(* IEC 61131-3 sources: AXOpen/src/components.rexroth.drives/ctrl/src/AxoCtrlxDriveXsc (part 4) *)

                IF _State>=UINT#430 AND _State<UINT#437 THEN
                    IF _AxisReference^.Data.Cycle <> MC_ReadBoolParameterCycle THEN
                        _AxisReference^.Data.Cycle := _AxisReference^.Data.Cycle - ULINT#1;
                        _State := UINT#439;
                    END_IF;
                END_IF;
            END_IF;

            IF NOT Enable AND MC_ReadBoolParameterEnable_PV AND _State>=UINT#430 AND _State<=UINT#439 THEN
                _AxisReference^.Status.CurrentMotionTaskId := AXOpen.Components.Drives.eAxoMotionTaskId#Axo_None;
                MC_ReadBoolParameterErrorID := WORD#0;
                MC_ReadBoolParameterCycle := ULINT#0;
                MC_ReadBoolParameterValid := FALSE;
                MC_ReadBoolParameterValue := FALSE;
                _State := UINT#0;
            END_IF;

            ErrorID := TO_DINT(MC_ReadBoolParameterErrorID);
            Valid := MC_ReadBoolParameterValid;
            Value := MC_ReadBoolParameterValue;
            MC_ReadBoolParameterEnable_PV := Enable;

        END_METHOD

        ///<summary>
        /// This method modifies the value of a vendor specific parameter.
        ///</summary>
        VAR INTERNAL
            MC_WriteParameterExecute_PV     : 	BOOL := FALSE;		//Enable - previous value
            MC_WriteParameterErrorID        : 	WORD;
            MC_WriteParameterCycle			: 	ULINT;
        END_VAR
        METHOD PUBLIC OVERRIDE MC_WriteParameter
            VAR_INPUT
                AxisRef         :   AXOpen.Components.Abstractions.Drives.IAxoAxisReference;
                Execute         :   BOOL;                       //  Write the value of the parameter at rising edge
                ParameterNumber :   DINT;                       //  Number of the parameter (correspondence between number andparameter is specified in the table above)
                Value           :   LINT;                       //  New value of the specified parameter
                ExecutionMode   :   AXOpen.Components.Abstractions.Drives.eAxoExecutionMode;          //  Defines the chronological sequence of the method.
            END_VAR
            VAR_OUTPUT
                Done            :   BOOL;                       //  Parameter successfully written
                Busy            :   BOOL;                       //  The method is not finished and new output values are to be expected.
                Error           :   BOOL;                       //  Signals that an error has occurred within the method
                ErrorID         :   DINT;                       //  Error identification
            END_VAR
            VAR
                _AxisReference :  REF_TO AXOpen.Components.Rexroth.Drives.AxoCtrlxDriveXscAxisReference;
            END_VAR

            _AxisReference ?= AxisRef;

            IF(_AxisReference = NULL) THEN
                Messenger.Activate(     UINT#1610, eAxoMessageCategory#ProgrammingError);
                DriveStatus.Error.Id := UINT#1610;
                RETURN;
            END_IF;

            IF THIS.AxoWriteParameter_Task.StartTriggered()  THEN
                _AxisReference^.Status.CurrentMotionTaskId := AXOpen.Components.Drives.eAxoMotionTaskId#Axo_WriteParameter;
            END_IF;

            IF Execute AND NOT MC_WriteParameterExecute_PV AND _State = UINT#0 THEN
                _AxisReference^.Data.Cycle := _AxisReference^.Data.Cycle + ULINT#2;
                MC_WriteParameterCycle := _AxisReference^.Data.Cycle ;
            END_IF;

            IF Execute THEN
                IF _State = UINT#0 THEN
                    Busy := TRUE;
                    THIS.CallTimers(FALSE);
                    DriveStatus.Error.Id :=  UINT#0;
                    TaskMessenger.Restore();
                    _State := UINT#440;
                END_IF;
                IF _State = UINT#440 THEN
                    IF _infoTimer.output THEN
                        TaskMessenger.Activate( UINT#640, eAxoMessageCategory#Potential);
                        DriveStatus.Error.Id := UINT#640;
                    END_IF;
                    Busy := TRUE;
                    _lword :=  TO_LWORD(Value);
                    _data8[0] := _lword.%B0;
                    _data8[1] := _lword.%B1;
                    _data8[2] := _lword.%B2;
                    _data8[3] := _lword.%B3;
                    _data8[4] := _lword.%B4;
                    _data8[5] := _lword.%B5;
                    _data8[6] := _lword.%B6;
                    _data8[7] := _lword.%B7;
                    _WriteRecord(   request     :=  TRUE,
                                    hardwareID  :=  (AxisRefExt.HWIDs.HW_S_0_0134_0_0),
                                    index       :=  ParameterNumber,
                                    length      :=  UINT#8,
                                    record      :=  _data8);
                    IF NOT _WriteRecord.busy AND _WriteRecord.done AND NOT _WriteRecord.error THEN
                        _State := UINT#441;
                    ElSIF _WriteRecord.error THEN
                        _WriteRecord(request := FALSE, record := _data8);
                        Messenger.Activate(         UINT#1611, eAxoMessageCategory#Error);
                        MC_WriteParameterErrorID := WORD#1611;
                        _State := UINT#449;
                    END_IF;
                END_IF;
                IF _State = UINT#441 THEN
                    _WriteRecord(request := FALSE, record := _data8);
                    IF NOT _WriteRecord.busy AND NOT _WriteRecord.done AND NOT _WriteRecord.error  THEN
                        _State := UINT#447;
                    END_IF;
                END_IF;
                IF _State = UINT#447 THEN
                    Done := TRUE;
                    MC_WriteParameterCycle := ULINT#0;
                END_IF;
                IF _State = UINT#449 THEN
                    MC_WriteParameterCycle := ULINT#0;
                    Error := TRUE;
                END_IF;

                IF _State>=UINT#440 AND _State<UINT#447 THEN
                    IF _AxisReference^.Data.Cycle <> MC_WriteParameterCycle THEN
                        _AxisReference^.Data.Cycle := _AxisReference^.Data.Cycle - ULINT#1;
                        _State := UINT#449;
                    END_IF;
                END_IF;
            END_IF;

            IF THIS.AxoWriteParameter_Task.DoneReached() AND _State>=UINT#440 AND _State<=UINT#449 THEN
                _AxisReference^.Status.CurrentMotionTaskId := AXOpen.Components.Drives.eAxoMotionTaskId#Axo_Done;
                MC_WriteParameterErrorID := WORD#0;
                // MC_WriteParameterCycle := ULINT#0;
                _State := UINT#0;
            END_IF;

            IF THIS.AxoWriteParameter_Task.RestoreTriggered() AND _State>=UINT#440 AND _State<=UINT#449 THEN
                _AxisReference^.Status.CurrentMotionTaskId := AXOpen.Components.Drives.eAxoMotionTaskId#Axo_None;
                MC_WriteParameterErrorID := WORD#0;
                MC_WriteParameterCycle := ULINT#0;
                _State := UINT#0;
            END_IF;

            ErrorID := TO_DINT(MC_WriteParameterErrorID);
            MC_WriteParameterExecute_PV := Execute;
        END_METHOD

        ///<summary>
        /// This method modifies the value of a vendor specific parameter of type Real.
        ///</summary>
        VAR INTERNAL
            MC_WriteRealParameterExecute_PV     : 	BOOL := FALSE;		//Enable - previous value
            MC_WriteRealParameterErrorID        : 	WORD;
            MC_WriteRealParameterCycle			: 	ULINT;
        END_VAR
        METHOD PUBLIC OVERRIDE MC_WriteRealParameter
            VAR_INPUT
                AxisRef         :   AXOpen.Components.Abstractions.Drives.IAxoAxisReference;
                Execute         :   BOOL;                       //  Write the value of the parameter at rising edge
                ParameterNumber :   DINT;                       //  Number of the parameter (correspondence between number andparameter is specified in the table above)
                Value           :   REAL;                       //  New value of the specified parameter
                ExecutionMode   :   AXOpen.Components.Abstractions.Drives.eAxoExecutionMode;          //  Defines the chronological sequence of the method.
            END_VAR
            VAR_OUTPUT
                Done            :   BOOL;                       //  Parameter successfully written
                Busy            :   BOOL;                       //  The method is not finished and new output values are to be expected.
                Error           :   BOOL;                       //  Signals that an error has occurred within the method
                ErrorID         :   DINT;                       //  Error identification
            END_VAR
            VAR
                _AxisReference :  REF_TO AXOpen.Components.Rexroth.Drives.AxoCtrlxDriveXscAxisReference;
            END_VAR

            _AxisReference ?= AxisRef;

            IF(_AxisReference = NULL) THEN
                Messenger.Activate(     UINT#1620, eAxoMessageCategory#ProgrammingError);
                DriveStatus.Error.Id := UINT#1620;
                RETURN;
            END_IF;

            IF THIS.AxoWriteRealParameter_Task.StartTriggered()  THEN
                _AxisReference^.Status.CurrentMotionTaskId := AXOpen.Components.Drives.eAxoMotionTaskId#Axo_WriteRealParameter;
            END_IF;

            IF Execute AND NOT MC_WriteRealParameterExecute_PV AND _State = UINT#0 THEN
                _AxisReference^.Data.Cycle := _AxisReference^.Data.Cycle + ULINT#2;
                MC_WriteRealParameterCycle := _AxisReference^.Data.Cycle ;
            END_IF;

            IF Execute THEN
                IF _State = UINT#0 THEN
                    Busy := TRUE;
                    _State := UINT#450;
                END_IF;
                IF _State = UINT#450 THEN
                    IF _infoTimer.output THEN
                        TaskMessenger.Activate( UINT#650, eAxoMessageCategory#Potential);
                        DriveStatus.Error.Id := UINT#650;
                    END_IF;
                    Busy := TRUE;
                    _dword :=  TO_DWORD(TO_DINT(Value));
                    _data4[0] := _dword.%B0;
                    _data4[1] := _dword.%B1;
                    _data4[2] := _dword.%B2;
                    _data4[3] := _dword.%B3;
                    _WriteRecord(   request     :=  TRUE,
                                    hardwareID  :=  (AxisRefExt.HWIDs.HW_S_0_0134_0_0),
                                    index       :=  ParameterNumber,
                                    length      :=  UINT#4,
                                    record      :=  _data4);
                    IF NOT _WriteRecord.busy AND _WriteRecord.done AND NOT _WriteRecord.error THEN
                        _State := UINT#451;
                    ElSIF _WriteRecord.error THEN
                        _WriteRecord(request := FALSE, record := _data4);
                        Messenger.Activate(             UINT#1621, eAxoMessageCategory#Error);
                        MC_WriteRealParameterErrorID := WORD#1621;
                        _State := UINT#459;
                    END_IF;
                END_IF;
                IF _State = UINT#451 THEN
                    IF _infoTimer.output THEN
                        TaskMessenger.Activate( UINT#651, eAxoMessageCategory#Potential);
                        DriveStatus.Error.Id := UINT#651;
                    END_IF;
                    Busy := TRUE;
                    _WriteRecord(request := FALSE, record := _data4);
                    IF NOT _WriteRecord.busy AND NOT _WriteRecord.done AND NOT _WriteRecord.error THEN
                        _State := UINT#457;
                    END_IF;
                END_IF;
                IF _State = UINT#457 THEN
                    Done := TRUE;
                    MC_WriteRealParameterCycle := ULINT#0;
                END_IF;
                IF _State = UINT#459 THEN
                    MC_WriteRealParameterCycle := ULINT#0;
                    Error := TRUE;
                END_IF;

                IF _State>=UINT#450 AND _State<UINT#457 THEN
                    IF _AxisReference^.Data.Cycle <> MC_WriteRealParameterCycle THEN
                        _AxisReference^.Data.Cycle := _AxisReference^.Data.Cycle - ULINT#1;
                        _State := UINT#459;
                    END_IF;
                END_IF;
            END_IF;

            IF THIS.AxoWriteRealParameter_Task.DoneReached() AND _State>=UINT#450 AND _State<=UINT#459 THEN
                _AxisReference^.Status.CurrentMotionTaskId := AXOpen.Components.Drives.eAxoMotionTaskId#Axo_Done;
                MC_WriteRealParameterErrorID := WORD#0;
                // MC_WriteRealParameterCycle := ULINT#0;
                _State := UINT#0;
            END_IF;

            IF THIS.AxoWriteRealParameter_Task.RestoreTriggered() AND _State>=UINT#450 AND _State<=UINT#459 THEN
                _AxisReference^.Status.CurrentMotionTaskId := AXOpen.Components.Drives.eAxoMotionTaskId#Axo_None;
                MC_WriteRealParameterErrorID := WORD#0;
                MC_WriteRealParameterCycle := ULINT#0;
                _State := UINT#0;
            END_IF;

            ErrorID := TO_DINT(MC_WriteRealParameterErrorID);
            MC_WriteRealParameterExecute_PV := Execute;
        END_METHOD

        ///<summary>
        /// This method modifies the value of a vendor specific parameter of type BOOL.
        ///</summary>
        VAR INTERNAL
            MC_WriteBoolParameterExecute_PV     : 	BOOL := FALSE;		//Enable - previous value
            MC_WriteBoolParameterErrorID        : 	WORD;
            MC_WriteBoolParameterCycle			: 	ULINT;
        END_VAR
        METHOD PUBLIC OVERRIDE MC_WriteBoolParameter
            VAR_INPUT
                AxisRef         :   AXOpen.Components.Abstractions.Drives.IAxoAxisReference;
                Execute         :   BOOL;                       //  Write the value of the parameter at rising edge
                ParameterNumber :   DINT;                       //  Number of the parameter (correspondence between number andparameter is specified in the table above)
                Value           :   BOOL;                       //  New value of the specified parameter
                ExecutionMode   :   AXOpen.Components.Abstractions.Drives.eAxoExecutionMode;          //  Defines the chronological sequence of the method.
            END_VAR
            VAR_OUTPUT
                Done            :   BOOL;                       //  Parameter successfully written
                Busy            :   BOOL;                       //  The method is not finished and new output values are to be expected.
                Error           :   BOOL;                       //  Signals that an error has occurred within the method
                ErrorID         :   DINT;                       //  Error identification
            END_VAR
            VAR
                _AxisReference :  REF_TO AXOpen.Components.Rexroth.Drives.AxoCtrlxDriveXscAxisReference;
            END_VAR

            _AxisReference ?= AxisRef;

            IF(_AxisReference = NULL) THEN
                Messenger.Activate(     UINT#1630, eAxoMessageCategory#ProgrammingError);
                DriveStatus.Error.Id := UINT#1630;
                RETURN;
            END_IF;

            IF THIS.AxoWriteBoolParameter_Task.StartTriggered()  THEN
                _AxisReference^.Status.CurrentMotionTaskId := AXOpen.Components.Drives.eAxoMotionTaskId#Axo_WriteBoolParameter;
            END_IF;

            IF Execute AND NOT MC_WriteBoolParameterExecute_PV AND _State = UINT#0 THEN
                _AxisReference^.Data.Cycle := _AxisReference^.Data.Cycle + ULINT#2;
                MC_WriteBoolParameterCycle := _AxisReference^.Data.Cycle ;
            END_IF;

            IF Execute THEN
                IF _State = UINT#0 THEN
                    Busy := TRUE;
                    _State := UINT#460;
                END_IF;
                IF _State = UINT#460 THEN
                    IF _infoTimer.output THEN
                        TaskMessenger.Activate( UINT#660, eAxoMessageCategory#Potential);
                        DriveStatus.Error.Id := UINT#660;
                    END_IF;
                    Busy := TRUE;
                    _dword :=  TO_DWORD(TO_DINT(Value));
                    _data2[0].%X0 := Value;
                    _WriteRecord(   request     :=  TRUE,
                                    hardwareID  :=  (AxisRefExt.HWIDs.HW_S_0_0134_0_0),
                                    index       :=  ParameterNumber,
                                    length      :=  UINT#2,
                                    record      :=  _data2);
                    IF NOT _WriteRecord.busy AND _WriteRecord.done AND NOT _WriteRecord.error THEN
                        _State := UINT#461;
                    ElSIF _WriteRecord.error THEN
                        _WriteRecord(request := FALSE, record := _data2);
                        Messenger.Activate(             UINT#1631, eAxoMessageCategory#Error);
                        MC_WriteBoolParameterErrorID := WORD#1631;
                        _State := UINT#469;
                    END_IF;
                END_IF;
                IF _State = UINT#461 THEN
                    IF _infoTimer.output THEN
                        TaskMessenger.Activate( UINT#661, eAxoMessageCategory#Potential);
                        DriveStatus.Error.Id := UINT#661;
                    END_IF;
                    Busy := TRUE;
                    _WriteRecord(request := FALSE, record := _data2);
                    IF NOT _WriteRecord.busy AND _WriteRecord.done AND NOT _WriteRecord.error THEN
                        _State := UINT#467;
                    END_IF;
                END_IF;
                IF _State = UINT#467 THEN
                    Done := TRUE;
                    MC_WriteBoolParameterCycle := ULINT#0;
                END_IF;
                IF _State = UINT#469 THEN
                    MC_WriteBoolParameterCycle := ULINT#0;
                    Error := TRUE;
                END_IF;

                IF _State>=UINT#460 AND _State<UINT#467 THEN
                    IF _AxisReference^.Data.Cycle <> MC_WriteBoolParameterCycle THEN
                        _AxisReference^.Data.Cycle := _AxisReference^.Data.Cycle - ULINT#1;
                        _State := UINT#469;
                    END_IF;
                END_IF;
            END_IF;

            IF THIS.AxoWriteBoolParameter_Task.DoneReached() AND _State>=UINT#460 AND _State<=UINT#469 THEN
                _AxisReference^.Status.CurrentMotionTaskId := AXOpen.Components.Drives.eAxoMotionTaskId#Axo_Done;
                MC_WriteBoolParameterErrorID := WORD#0;
                // MC_WriteBoolParameterCycle := ULINT#0;
                _State := UINT#0;
            END_IF;

            IF THIS.AxoWriteBoolParameter_Task.RestoreTriggered() AND _State>=UINT#460 AND _State<=UINT#469 THEN
                _AxisReference^.Status.CurrentMotionTaskId := AXOpen.Components.Drives.eAxoMotionTaskId#Axo_None;
                MC_WriteBoolParameterErrorID := WORD#0;
                MC_WriteBoolParameterCycle := ULINT#0;
                _State := UINT#0;
            END_IF;

            ErrorID := TO_DINT(MC_WriteBoolParameterErrorID);
            MC_WriteBoolParameterExecute_PV := Execute;
        END_METHOD

        ///<summary>
        /// This method gives access to the value of the input, referenced by the datatype MC_INPUT_REF.
        /// It provides the value of the referenced input (BOOL).
        ///</summary>
        VAR INTERNAL
            MC_ReadDigitalInputEnable_PV        : 	BOOL := FALSE;		//Enable - previous value
            MC_ReadDigitalInputErrorID          : 	WORD;
            MC_ReadDigitalInputCycle			: 	ULINT;
            MC_ReadDigitalInputValue			: 	BOOL;
            MC_ReadDigitalInputValid			: 	BOOL;
        END_VAR
        METHOD PUBLIC OVERRIDE MC_ReadDigitalInput
            VAR_INPUT
                AxisRef         :   AXOpen.Components.Abstractions.Drives.IAxoAxisReference;
                Enable          :   BOOL;                       //  Get the value of the selected input signal continuously while enabled
                InputNumber     :   INT;                        //  Selects the input. Can be part of MC_INPUT_REF, if only one single input is referenced.
            END_VAR
            VAR_OUTPUT
                Valid           :   BOOL;                       //  A valid output is available at the method
                Busy            :   BOOL;                       //  The method is not finished and new output values are to be expected
                Error           :   BOOL;                       //  Signals that an error has occurred within the method
                ErrorID         :   DINT;                       //  Error identification
                Value           :   BOOL;                       //  The value of the selected input signal
            END_VAR
            VAR
                _AxisReference :  REF_TO AXOpen.Components.Rexroth.Drives.AxoCtrlxDriveXscAxisReference;
            END_VAR

            _AxisReference ?= AxisRef;

            IF(_AxisReference = NULL) THEN
                Messenger.Activate(     UINT#1640, eAxoMessageCategory#ProgrammingError);
                DriveStatus.Error.Id := UINT#1640;
                RETURN;
            END_IF;

            IF(InputNumber < 0 OR InputNumber >256) THEN   //  TODO check the min max input number
                Messenger.Activate(     UINT#1641, eAxoMessageCategory#ProgrammingError);
                DriveStatus.Error.Id := UINT#1641;
                RETURN;
            END_IF;

            IF Enable AND NOT MC_ReadDigitalInputEnable_PV AND _State = UINT#0 THEN
                _AxisReference^.Status.CurrentMotionTaskId := AXOpen.Components.Drives.eAxoMotionTaskId#Axo_ReadDigitalInput;
                _AxisReference^.Data.Cycle := _AxisReference^.Data.Cycle + ULINT#2;
                MC_ReadDigitalInputCycle := _AxisReference^.Data.Cycle ;
            END_IF;

            IF Enable THEN
                IF _State = UINT#0 THEN
                    Busy := TRUE;
                    MC_ReadDigitalInputErrorID := WORD#16#0000;
                    _State := UINT#470;
                END_IF;
                IF _State = UINT#470 THEN
                    IF _infoTimer.output THEN
                        TaskMessenger.Activate( UINT#670, eAxoMessageCategory#Potential);
                        DriveStatus.Error.Id := UINT#670;
                    END_IF;
                    Busy := TRUE;
                    _ReadRecord(    request     :=  TRUE,
                                    hardwareID          :=  (AxisRefExt.HWIDs.HW_S_0_0134_0_0),
                                    index       :=  DINT#4403, //P-0-0307.0.0  16#1000 + 307 = 4096+307=4403
                                    maxLength   :=  UINT#4,
                                    record      :=  _data4);
                    IF NOT _ReadRecord.busy AND _ReadRecord.valid AND NOT _ReadRecord.error THEN
                        _dword.%B0   :=  _data4[0];
                        _dword.%B1   :=  _data4[1];
                        _dword.%B2   :=  _data4[2];
                        _dword.%B3   :=  _data4[3];
                        MC_ReadDigitalInputValid := TRUE;
                        MC_ReadDigitalInputValue := System.BitAccess.GetBit(_dword, TO_USINT(InputNumber));
                        _State := UINT#471;
                    END_IF;
                    IF _ReadRecord.error THEN
                        _ReadRecord(request := FALSE, record := _data4);
                        Messenger.Activate(             UINT#1642, eAxoMessageCategory#Error);
                        MC_ReadDigitalInputErrorID :=   WORD#1642;
                        _State := UINT#479;
                    END_IF;
                END_IF;
                IF _State = UINT#471 THEN
                    IF _infoTimer.output THEN
                        TaskMessenger.Activate( UINT#671, eAxoMessageCategory#Potential);
                        DriveStatus.Error.Id := UINT#671;
                    END_IF;
                    Busy := TRUE;
                    _ReadRecord(request := FALSE, record := _data4);
                    IF NOT _ReadRecord.busy AND NOT _ReadRecord.valid AND NOT _ReadRecord.error  THEN
                        _State := UINT#470;
                    END_IF;
                END_IF;
                IF _State = UINT#479 THEN
                    Error := TRUE;
                END_IF;

                IF _State>=UINT#470 AND _State<UINT#477 THEN
                    IF _AxisReference^.Data.Cycle <> MC_ReadDigitalInputCycle THEN
                        _AxisReference^.Data.Cycle := _AxisReference^.Data.Cycle - ULINT#1;
                        _State := UINT#479;
                    END_IF;
                END_IF;
            END_IF;

            IF NOT Enable AND MC_ReadDigitalInputEnable_PV AND _State>=UINT#470 AND _State<=UINT#479 THEN
                _AxisReference^.Status.CurrentMotionTaskId := AXOpen.Components.Drives.eAxoMotionTaskId#Axo_None;
                MC_ReadDigitalInputErrorID := WORD#0;
                MC_ReadDigitalInputCycle := ULINT#0;
                MC_ReadDigitalInputValid := FALSE;
                MC_ReadDigitalInputValue := FALSE;
                _State := UINT#0;
            END_IF;

            ErrorID := TO_DINT(MC_ReadDigitalInputErrorID);
            Valid := MC_ReadDigitalInputValid;
            Value := MC_ReadDigitalInputValue;
            MC_ReadDigitalInputEnable_PV := Enable;
        END_METHOD

        ///<summary>
        /// This method provides access to the value of a digital output, referenced by the datatype MC_OUTPUT_REF.
        /// It provides the value of the referenced output (BOOL).
        ///</summary>
        VAR INTERNAL
            MC_ReadDigitalOutputEnable_PV        : 	BOOL := FALSE;		//Enable - previous value
            MC_ReadDigitalOutputErrorID          : 	WORD;
            MC_ReadDigitalOutputCycle			: 	ULINT;
            MC_ReadDigitalOutputValue			: 	BOOL;
            MC_ReadDigitalOutputValid			: 	BOOL;
        END_VAR
        METHOD PUBLIC OVERRIDE MC_ReadDigitalOutput
            VAR_INPUT
                AxisRef         :   AXOpen.Components.Abstractions.Drives.IAxoAxisReference;
                Enable          :   BOOL;                       //  Get the value of the selected output signal continuously while enabled
                OutputNumber    :   INT;                        //  Selects the output. Can be part of MC_OUTPUT_REF, if only one single output is referenced.
            END_VAR
            VAR_OUTPUT
                Valid           :   BOOL;                       //  A valid output is available at the method
                Busy            :   BOOL;                       //  The method is not finished and new output values are to be expected
                Error           :   BOOL;                       //  Signals that an error has occurred within the method
                ErrorID         :   DINT;                       //  Error identification
                Value           :   BOOL;                       //  The value of the selected output signal
            END_VAR
            VAR
                _AxisReference :  REF_TO AXOpen.Components.Rexroth.Drives.AxoCtrlxDriveXscAxisReference;
            END_VAR

            _AxisReference ?= AxisRef;

            IF(_AxisReference = NULL) THEN
                Messenger.Activate(     UINT#1650, eAxoMessageCategory#ProgrammingError);
                DriveStatus.Error.Id := UINT#1650;
                RETURN;
            END_IF;

            IF(OutputNumber < 0 OR OutputNumber >256) THEN   //  TODO check the min max input number
                Messenger.Activate(     UINT#1651, eAxoMessageCategory#ProgrammingError);
                DriveStatus.Error.Id := UINT#1651;
                RETURN;
            END_IF;

            IF Enable AND NOT MC_ReadDigitalOutputEnable_PV AND _State = UINT#0 THEN
                _AxisReference^.Status.CurrentMotionTaskId := AXOpen.Components.Drives.eAxoMotionTaskId#Axo_ReadDigitalOutput;
                _AxisReference^.Data.Cycle := _AxisReference^.Data.Cycle + ULINT#2;
                MC_ReadDigitalOutputCycle := _AxisReference^.Data.Cycle ;
            END_IF;

            IF Enable THEN
                IF _State = UINT#0 THEN
                    Busy := TRUE;
                    MC_ReadDigitalOutputErrorID := WORD#16#0000;
                    _State := UINT#480;
                END_IF;
                IF _State = UINT#480 THEN
                    IF _infoTimer.output THEN
                        TaskMessenger.Activate( UINT#680, eAxoMessageCategory#Potential);
                        DriveStatus.Error.Id := UINT#680;
                    END_IF;
                    Busy := TRUE;
                    _ReadRecord(    request     :=  TRUE,
                                    hardwareID          :=  (AxisRefExt.HWIDs.HW_S_0_0134_0_0),
                                    index       :=  DINT#4409, //P-0-0313.0.0  16#1000 + 313 = 4096+313=4409
                                    maxLength   :=  UINT#4,
                                    record      :=  _data4);
                    IF NOT _ReadRecord.busy AND _ReadRecord.valid AND NOT _ReadRecord.error THEN
                        _dword.%B0   :=  _data4[0];
                        _dword.%B1   :=  _data4[1];
                        _dword.%B2   :=  _data4[2];
                        _dword.%B3   :=  _data4[3];
                        MC_ReadDigitalOutputValid := TRUE;
                        MC_ReadDigitalOutputValue := System.BitAccess.GetBit(_dword, TO_USINT(OutputNumber));
                        _State := UINT#481;
                    END_IF;
                    IF _ReadRecord.error THEN
                        _ReadRecord(request := FALSE, record := _data4);
                        Messenger.Activate(             UINT#1652, eAxoMessageCategory#Error);
                        MC_ReadDigitalOutputErrorID :=  WORD#1652;
                        _State := UINT#489;
                    END_IF;
                END_IF;
                IF _State = UINT#481 THEN
                    IF _infoTimer.output THEN
                        TaskMessenger.Activate( UINT#681, eAxoMessageCategory#Potential);
                        DriveStatus.Error.Id := UINT#681;
                    END_IF;
                    Busy := TRUE;
                    _ReadRecord(request := FALSE, record := _data4);
                    IF NOT _ReadRecord.busy AND NOT _ReadRecord.valid AND NOT _ReadRecord.error  THEN
                        _State := UINT#480;
                    END_IF;
                END_IF;
                IF _State = UINT#489 THEN
                    Error := TRUE;
                END_IF;

                IF _State>=UINT#480 AND _State<UINT#487 THEN
                    IF _AxisReference^.Data.Cycle <> MC_ReadDigitalOutputCycle THEN
                        _AxisReference^.Data.Cycle := _AxisReference^.Data.Cycle - ULINT#1;
                        _State := UINT#489;
                    END_IF;
                END_IF;
            END_IF;

            IF NOT Enable AND MC_ReadDigitalOutputEnable_PV AND _State>=UINT#480 AND _State<=UINT#489 THEN
                _AxisReference^.Status.CurrentMotionTaskId := AXOpen.Components.Drives.eAxoMotionTaskId#Axo_None;
                MC_ReadDigitalOutputErrorID := WORD#0;
                MC_ReadDigitalOutputCycle := ULINT#0;
                MC_ReadDigitalOutputValid := FALSE;
                MC_ReadDigitalOutputValue := FALSE;
                _State := UINT#0;
            END_IF;

            ErrorID := TO_DINT(MC_ReadDigitalOutputErrorID);
            Valid := MC_ReadDigitalOutputValid;
            Value := MC_ReadDigitalOutputValue;
            MC_ReadDigitalOutputEnable_PV := Enable;
        END_METHOD

        ///<summary>
        /// This method writes a value to the output referenced by the argument ‘Output’ once (with rising edge of Execute)
        ///</summary>
        VAR INTERNAL
            MC_WriteDigitalOutputExecute_PV     : 	BOOL := FALSE;		//Enable - previous value
            MC_WriteDigitalOutputErrorID        : 	WORD;
            MC_WriteDigitalOutputCycle			: 	ULINT;
            MC_WriteDigitalOutputParameterPV    : 	DWORD;
        END_VAR
        METHOD PUBLIC OVERRIDE MC_WriteDigitalOutput
            VAR_INPUT
                AxisRef         :   AXOpen.Components.Abstractions.Drives.IAxoAxisReference;
                Execute         :   BOOL;                       //  Write the value of the selected output
                OutputNumber    :   INT;                        //  Selects the output. Can be part of MC_OUTPUT_REF, if only one single output is referenced.
                Value           :   BOOL;                       //  The value of the selected output signal
                ExecutionMode   :   AXOpen.Components.Abstractions.Drives.eAxoExecutionMode;          //  Defines the chronological sequence of the method.
            END_VAR
            VAR_OUTPUT
                Done            :   BOOL;                       //  Writing of the output signal value is done
                Busy            :   BOOL;                       //  The method is not finished and new output values are to be expected.
                Error           :   BOOL;                       //  Signals that an error has occurred within the method
                ErrorID         :   DINT;                       //  Error identification
            END_VAR
            VAR
                _AxisReference  :  REF_TO AXOpen.Components.Rexroth.Drives.AxoCtrlxDriveXscAxisReference;
                Valid_          :   BOOL;
                Error_          :   BOOL;
                ErrorID_        :   WORD;
            END_VAR

            _AxisReference ?= AxisRef;

            IF(_AxisReference = NULL) THEN
                Messenger.Activate(     UINT#1660, eAxoMessageCategory#ProgrammingError);
                DriveStatus.Error.Id := UINT#1660;
                RETURN;
            END_IF;

            IF(OutputNumber < 0 OR OutputNumber >256) THEN   //  TODO check the min max input number
                Messenger.Activate(     UINT#1661, eAxoMessageCategory#ProgrammingError);
                DriveStatus.Error.Id := UINT#1661;
                RETURN;
            END_IF;

            IF THIS.AxoWriteDigitalOutput_Task.StartTriggered()  THEN
                _AxisReference^.Status.CurrentMotionTaskId := AXOpen.Components.Drives.eAxoMotionTaskId#Axo_WriteDigitalOutput;
            END_IF;

            IF Execute AND NOT MC_WriteDigitalOutputExecute_PV AND _State = UINT#0 THEN
                _AxisReference^.Data.Cycle := _AxisReference^.Data.Cycle + ULINT#2;
                MC_WriteDigitalOutputCycle := _AxisReference^.Data.Cycle ;
            END_IF;

            IF Execute THEN
                IF _State = UINT#0 THEN
                    Busy := TRUE;
                    _State := UINT#490;
                END_IF;
                IF _State = UINT#490 THEN
                    IF _infoTimer.output THEN
                        TaskMessenger.Activate( UINT#690, eAxoMessageCategory#Potential);
                        DriveStatus.Error.Id := UINT#690;
                    END_IF;
                    Busy := TRUE;
                    _ReadRecord(    request     :=  TRUE,
                                    hardwareID          :=  (AxisRefExt.HWIDs.HW_S_0_0134_0_0),
                                    index       :=  DINT#4409, //P-0-0313.0.0  16#1000 + 313 = 4096+313=4409
                                    maxLength   :=  UINT#4,
                                    record      :=  _data4);
                    IF NOT _ReadRecord.busy AND _ReadRecord.valid AND NOT _ReadRecord.error THEN
                        MC_WriteDigitalOutputParameterPV.%B0   :=  _data4[0];
                        MC_WriteDigitalOutputParameterPV.%B1   :=  _data4[1];
                        MC_WriteDigitalOutputParameterPV.%B2   :=  _data4[2];
                        MC_WriteDigitalOutputParameterPV.%B3   :=  _data4[3];
                        _State := UINT#491;
                    END_IF;
                    IF  _ReadRecord.error THEN
                        Messenger.Activate(             UINT#1662, eAxoMessageCategory#Error);
                        MC_WriteDigitalOutputErrorID := WORD#1662;
                        _State := UINT#499;
                    END_IF;
                END_IF;
                IF _State = UINT#491 THEN
                    IF _infoTimer.output THEN
                        TaskMessenger.Activate( UINT#691, eAxoMessageCategory#Potential);
                        DriveStatus.Error.Id := UINT#691;
                    END_IF;
                    Busy := TRUE;
                    _ReadRecord(request := FALSE, record := _data8);
                    IF NOT _ReadRecord.busy AND NOT _ReadRecord.valid AND NOT _ReadRecord.error  THEN
                        _State := UINT#492;
                    END_IF;
                END_IF;
                IF _State = UINT#492 THEN
                    IF _infoTimer.output THEN
                        TaskMessenger.Activate( UINT#692, eAxoMessageCategory#Potential);
                        DriveStatus.Error.Id := UINT#692;
                    END_IF;
                    Busy := TRUE;
                    MC_WriteDigitalOutputParameterPV := System.BitAccess.SetBit(value := MC_WriteDigitalOutputParameterPV,bitValue := Value,index := TO_USINT(OutputNumber));
                    _State := UINT#493;
                END_IF;
                IF _State = UINT#493 THEN
                    Busy := TRUE;
                    _data4[0] := MC_WriteDigitalOutputParameterPV.%B0;
                    _data4[1] := MC_WriteDigitalOutputParameterPV.%B1;
                    _data4[2] := MC_WriteDigitalOutputParameterPV.%B2;
                    _data4[3] := MC_WriteDigitalOutputParameterPV.%B3;
                    _WriteRecord(   request     :=  TRUE,
                                    hardwareID  :=  (AxisRefExt.HWIDs.HW_S_0_0134_0_0),
                                    index       :=  DINT#4409, //P-0-0313.0.0  16#1000 + 313 = 4096+313=4409
                                    length      :=  UINT#4,
                                    record      :=  _data4);
                    IF NOT _WriteRecord.busy AND _WriteRecord.done AND NOT _WriteRecord.error THEN
                        _State := UINT#494;
                    ElSIF _WriteRecord.error THEN
                        _WriteRecord(request := FALSE, record := _data4);
                        Messenger.Activate(         UINT#1663, eAxoMessageCategory#Error);
                        MC_WriteParameterErrorID := WORD#1663;
                        _State := UINT#499;
                    END_IF;
                END_IF;
                IF _State = UINT#494 THEN
                    _WriteRecord(request := FALSE, record := _data4);
                    IF NOT _WriteRecord.busy AND NOT _WriteRecord.done AND NOT _WriteRecord.error  THEN
                        _State := UINT#497;
                    END_IF;
                END_IF;

                IF _State = UINT#497 THEN
                    Done := TRUE;
                    MC_WriteDigitalOutputCycle := ULINT#0;
                END_IF;
                IF _State = UINT#499 THEN
                    MC_WriteDigitalOutputCycle := ULINT#0;
                    Error := TRUE;
                END_IF;

                IF _State>=UINT#490 AND _State<UINT#497 THEN
                    IF _AxisReference^.Data.Cycle <> MC_WriteDigitalOutputCycle THEN
                        _AxisReference^.Data.Cycle := _AxisReference^.Data.Cycle - ULINT#1;
                        _State := UINT#499;
                    END_IF;
                END_IF;
            END_IF;

            IF THIS.AxoWriteDigitalOutput_Task.DoneReached() AND _State>=UINT#490 AND _State<=UINT#499 THEN
                _AxisReference^.Status.CurrentMotionTaskId := AXOpen.Components.Drives.eAxoMotionTaskId#Axo_Done;
                MC_WriteDigitalOutputErrorID := WORD#0;
                // MC_WriteDigitalOutputCycle := ULINT#0;
                _State := UINT#0;
            END_IF;

            IF THIS.AxoWriteDigitalOutput_Task.RestoreTriggered() AND _State>=UINT#490 AND _State<=UINT#499 THEN
                _AxisReference^.Status.CurrentMotionTaskId := AXOpen.Components.Drives.eAxoMotionTaskId#Axo_None;
                MC_WriteDigitalOutputErrorID := WORD#0;
                MC_WriteDigitalOutputCycle := ULINT#0;
                _State := UINT#0;
            END_IF;

            ErrorID := TO_DINT(MC_WriteDigitalOutputErrorID);
            MC_WriteDigitalOutputExecute_PV := Execute;

        END_METHOD

        ///<summary>
        /// This method returns the actual position.
        ///<summary>
        METHOD PUBLIC OVERRIDE MC_ReadActualPosition
             VAR_INPUT
                AxisRef         :   AXOpen.Components.Abstractions.Drives.IAxoAxisReference;
                Enable          :   BOOL;                       //  Get the value of the parameter continuously while enabled
            END_VAR
            VAR_OUTPUT
                Valid           :   BOOL;                       //  A valid output is available at the method
                Busy            :   BOOL;                       //  The method is not finished and new output values are to be expected
                Error           :   BOOL;                       //  Signals that an error has occurred within the method
                ErrorID         :   DINT;                       //  Error identification
                Position        :   LREAL;                       //  New absolute position (in axis’ unit [u])
            END_VAR
            VAR
                _AxisReference :  REF_TO AXOpen.Components.Rexroth.Drives.AxoCtrlxDriveXscAxisReference;
            END_VAR

            _AxisReference ?= AxisRef;

            IF(_AxisReference = NULL) THEN
                Messenger.Activate(     UINT#1670, eAxoMessageCategory#ProgrammingError);
                DriveStatus.Error.Id := UINT#1670;
                RETURN;
            END_IF;

            IF Enable THEN
                Valid := TRUE;
                Position := THIS.ActualPosition;
            END_IF;
        END_METHOD

        ///<summary>
        /// This method returns the value of the actual velocity as long as ‘Enable’ is set. ‘Valid’ is true when the
        /// dataoutput ‘Velocity’ is valid. If ‘Enable’ is Reset, the data loses its validity, and all outputs are reset,
        /// no matter if new data is available.
        ///<summary>
        METHOD PUBLIC OVERRIDE MC_ReadActualVelocity
            VAR_INPUT
                AxisRef         :   AXOpen.Components.Abstractions.Drives.IAxoAxisReference;
                Enable          :   BOOL;                       //  Get the value of the parameter continuously while enabled
            END_VAR
            VAR_OUTPUT
                Valid           :   BOOL;                       //  A valid output is available at the method
                Busy            :   BOOL;                       //  The method is not finished and new output values are to be expected
                Error           :   BOOL;                       //  Signals that an error has occurred within the method
                ErrorID         :   DINT;                       //  Error identification
                Velocity        :   LREAL;                       //  The value of the actual velocity (in axis’ unit [u/s])
            END_VAR
            VAR
                _AxisReference :  REF_TO AXOpen.Components.Rexroth.Drives.AxoCtrlxDriveXscAxisReference;
            END_VAR

            _AxisReference ?= AxisRef;

            IF(_AxisReference = NULL) THEN
                Messenger.Activate(     UINT#1680, eAxoMessageCategory#ProgrammingError);
                DriveStatus.Error.Id := UINT#1680;
                RETURN;
            END_IF;

            IF Enable THEN
                Valid := TRUE;
                Velocity := THIS.ActualVelocity;
            END_IF;
        END_METHOD

        ///<summary>
        /// This method returns the value of the actual torque or force as long as ‘Enable’ is set. ‘Valid’ is true when the
        /// data-output ‘Torque’ is valid. If ‘Enable’ is Reset, the data loses its validity, and ‘Valid’ is also reset,
        /// no matter if new data is available.
        ///<summary>
        METHOD PUBLIC OVERRIDE MC_ReadActualTorque
            VAR_INPUT
                AxisRef         :   AXOpen.Components.Abstractions.Drives.IAxoAxisReference;
                Enable          :   BOOL;                       //  Get the value of the parameter continuously while enabled
            END_VAR
            VAR_OUTPUT
                Valid           :   BOOL;                       //  A valid output is available at the method
                Busy            :   BOOL;                       //  The method is not finished and new output values are to be expected
                Error           :   BOOL;                       //  Signals that an error has occurred within the method
                ErrorID         :   DINT;                       //  Error identification
                Torque          :   LREAL;                       //  The value of the actual torque or force (in technical units)
            END_VAR
            VAR
                _AxisReference :  REF_TO AXOpen.Components.Rexroth.Drives.AxoCtrlxDriveXscAxisReference;
            END_VAR

            _AxisReference ?= AxisRef;

            IF(_AxisReference = NULL) THEN
                Messenger.Activate(     UINT#1690, eAxoMessageCategory#ProgrammingError);
                DriveStatus.Error.Id := UINT#1690;
                RETURN;
            END_IF;

            IF Enable THEN
                Valid := TRUE;
                Torque := THIS.ActualTorque;
            END_IF;
        END_METHOD

        ///<summary>
        /// This method returns in detail the status of the State diagram of the axis
        ///</summary>
        VAR INTERNAL
            MC_ReadStatusEnable_PV				: 	BOOL := FALSE;		//Enable - previous value
            MC_ReadStatusDone_PV				:	BOOL := FALSE;		//Done - previous value
            MC_ReadStatusStateNumber			: 	INT; 				//Call number of the method MC_ReadRealParameter
        END_VAR
        METHOD PUBLIC OVERRIDE MC_ReadStatus
            VAR_INPUT
                AxisRef             :   AXOpen.Components.Abstractions.Drives.IAxoAxisReference;
                Enable              :   BOOL;                       //  Get the value of the parameter continuously while enabled
            END_VAR
            VAR_OUTPUT
                Valid               :   BOOL;                       //  A valid output is available at the method
                Busy                :   BOOL;                       //  The method is not finished and new output values are to be expected
                Error               :   BOOL;                       //  Signals that an error has occurred within the method
                ErrorID             :   DINT;                       //  Error identification
                ErrorStop           :   BOOL;                       //  See_State diagram
                Disabled            :   BOOL;                       //  See_State diagram
                Stopping            :   BOOL;                       //  See_State diagram
                Homing              :   BOOL;                       //  See_State diagram
                Standstill          :   BOOL;                       //  See_State diagram
                DiscreteMotion      :   BOOL;                       //  See_State diagram
                ContinuousMotion     :   BOOL;                       //  See_State diagram
                SynchronizedMotion  : BOOL;                       //  See_State diagram
            END_VAR
            VAR
                _AxisReference :  REF_TO AXOpen.Components.Rexroth.Drives.AxoCtrlxDriveXscAxisReference;
            END_VAR

            _AxisReference ?= AxisRef;

            IF(_AxisReference = NULL) THEN
                Messenger.Activate(     UINT#1700, eAxoMessageCategory#ProgrammingError);
                DriveStatus.Error.Id := UINT#1700;
                RETURN;
            END_IF;

            // IF Enable THEN
            //     THIS.UpdateInputs(_AxisReference^);
            //     Valid := TRUE;
            //     Error                   := _AxisReference^.Telegram111_In.ZSW1.faultPresent;
            //     ErrorID                 := TO_WORD(_AxisReference^.Telegram111_In.Fault_Code);
            //     ErrorStop               := DriveState = AXOpen.Components.Drives.eAxoDriveState#ErrorStop;;
            //     Disabled                := DriveState = AXOpen.Components.Drives.eAxoDriveState#Disabled;
            //     Stopping                := DriveState = AXOpen.Components.Drives.eAxoDriveState#Stopping;
            //     Homing                  := DriveState = AXOpen.Components.Drives.eAxoDriveState#Homing;
            //     Standstill              := DriveState = AXOpen.Components.Drives.eAxoDriveState#Standstill;
            //     DiscreteMotion          := DriveState = AXOpen.Components.Drives.eAxoDriveState#DiscreteMotion;
            //     ContinuousMotion        := DriveState = AXOpen.Components.Drives.eAxoDriveState#ContinuousMotion;
            //     SynchronizedMotion      := DriveState = AXOpen.Components.Drives.eAxoDriveState#SynchronizedMotion;
            // END_IF;
        END_METHOD

        ///<summary>
        /// This method returns in detail the status of the axis with respect to the motion currently in progress.
        ///</summary>
        VAR INTERNAL
            MC_ReadMotionStateEnable_PV     : 	BOOL := FALSE;		//Enable - previous value
            MC_ReadMotionStateErrorID       : 	WORD;
            MC_ReadMotionStateCycle			: 	ULINT;
            MC_ReadMotionStateValue			: 	LINT;
            MC_ReadMotionStateValid			: 	BOOL;
        END_VAR
        METHOD PUBLIC OVERRIDE MC_ReadMotionState
            VAR_INPUT
                AxisRef         :   AXOpen.Components.Abstractions.Drives.IAxoAxisReference;
                Enable          :   BOOL;                       //  Get the value of the parameter continuously while enabled
                Source          :   AXOpen.Components.Abstractions.Drives.eAxoSource;                 //  Defines the source of the relevant data: CommandedValue;SetValue, ActualValue.
            END_VAR
            VAR_OUTPUT
                Valid           :   BOOL;                       //  A valid output is available at the method
                Busy            :   BOOL;                       //  The method is not finished and new output values are to be expected
                Error           :   BOOL;                       //  Signals that an error has occurred within the method
                ErrorID         :   DINT;                       //  Error identification
                ConstantVelocity:   BOOL;                       //  Velocity is constant. Velocity may be 0. For the actual value a window is applicable (window is vendor specific)
                Accelerating    :   BOOL;                       //  Increasing the absolute value of the velocity
                Decelerating    :   BOOL;                       //  Decreasing the absolute value of the velocity
                DirectionPositive:  BOOL;                       //  Signals that the position is increasing
                DirectionNegative:  BOOL;                       //  Signals that the position is decreasing
            END_VAR
            VAR
                _AxisReference :  REF_TO AXOpen.Components.Rexroth.Drives.AxoCtrlxDriveXscAxisReference;
            END_VAR

            _AxisReference ?= AxisRef;

            IF(_AxisReference = NULL) THEN
                Messenger.Activate(     UINT#1710, eAxoMessageCategory#ProgrammingError);
                DriveStatus.Error.Id := UINT#1710;
                RETURN;
            END_IF;

            // IF Enable THEN
            //     THIS.UpdateInputs(_AxisReference^);
            //     Valid := TRUE;
            //     Error                   := _AxisReference^.Telegram111_In.ZSW1.faultPresent;
            //     ErrorID                 := TO_WORD(_AxisReference^.Telegram111_In.Fault_Code);
            //     ConstantVelocity        := FALSE;
            //     Accelerating            := _AxisReference^.Telegram111_In.ZSW1.axisAccelerates;
            //     Decelerating            := _AxisReference^.Telegram111_In.ZSW1.axisDecelerates;
            //     DirectionPositive       := _AxisReference^.Telegram111_In.POS_ZSW2.%X4;
            //     DirectionNegative       := _AxisReference^.Telegram111_In.POS_ZSW2.%X5;
            //  END_IF;
        END_METHOD

        ///<summary>
        /// This method reads information concerning an axis, like modes, inputs directly related to the axis,
        /// and certain status information.
        ///<summary>
        METHOD PUBLIC OVERRIDE MC_ReadAxisInfo
            VAR_INPUT
                AxisRef             :   AXOpen.Components.Abstractions.Drives.IAxoAxisReference;
                Enable              :   BOOL;                       //  Get the value of the parameter continuously while enabled
            END_VAR
            VAR_OUTPUT
                Valid               :   BOOL;                       //  A valid output is available at the method
                Busy                :   BOOL;                       //  The method is not finished and new output values are to be expected
                Error               :   BOOL;                       //  Signals that an error has occurred within the method
                ErrorID             :   DINT;                       //  Error identification
                HomeAbsSwitch       :   BOOL;                       //  Digital home switch input is active
                LimitSwitchPos      :   BOOL;                       //  Positive hardware end switch is active
                LimitSwitchNeg      :   BOOL;                       //  Negative hardware end switch is active
                Simulation          :   BOOL;                       //  Axis is in simulation mode (e.g. motor is simulated)
                CommunicationReady  :   BOOL;                       //  “Network” is initialized and ready for communication
                ReadyForPowerOn     :   BOOL;                       //  Drive is ready to be enabled (power on)
                PowerOn             :   BOOL;                       //  If TRUE shows that the power stage is switched ON
                IsHomed             :   BOOL;                       //  The absolute reference position is known for the axis (axis is homed)
                AxisWarning         :   BOOL;                       //  Warning(s) on the axis is present
            END_VAR
            VAR
                _AxisReference :  REF_TO AXOpen.Components.Rexroth.Drives.AxoCtrlxDriveXscAxisReference;
            END_VAR

            _AxisReference ?= AxisRef;

            IF(_AxisReference = NULL) THEN
                Messenger.Activate(     UINT#1720, eAxoMessageCategory#ProgrammingError);
                DriveStatus.Error.Id := UINT#1720;
                RETURN;
            END_IF;

            // IF Enable THEN
            //     THIS.UpdateInputs(_AxisReference^);
            //     Valid := TRUE;
            //     Error                   := _AxisReference^.Telegram111_In.ZSW1.faultPresent;
            //     ErrorID                 := TO_WORD(_AxisReference^.Telegram111_In.Fault_Code);
            //     HomeAbsSwitch           := FALSE;
            //     LimitSwitchPos          := _AxisReference^.Telegram111_In.POS_ZSW1.%X9;
            //     LimitSwitchNeg          := _AxisReference^.Telegram111_In.POS_ZSW1.%X8;
            //     Simulation              := FALSE;
            //     CommunicationReady      := FALSE;
            //     ReadyForPowerOn         := _AxisReference^.Telegram111_In.ZSW1.readyForSwitchOn;
            //     PowerOn                 := _AxisReference^.Telegram111_In.ZSW1.operationEnabled;
            //     IsHomed                 := _AxisReference^.Telegram111_In.ZSW1.homePosSet;
            //     AxisWarning             := _AxisReference^.Telegram111_In.ZSW1.warningActive;
            // END_IF;
        END_METHOD

        ///<summary>
        /// This method presents general axis errors not relating to the methods.
        /// (for instance axis errors, drive errors, communication errors)
        ///</summary>
        VAR INTERNAL
            MC_ReadAxisErrorEnable_PV        : 	BOOL := FALSE;		//Enable - previous value
            MC_ReadAxisErrorErrorID          : 	WORD;
            MC_ReadAxisErrorCycle			: 	ULINT;
            MC_ReadAxisErrorValue			: 	LINT;
            MC_ReadAxisErrorValid			: 	BOOL;
            LastMessageCode :   ULINT;
        END_VAR
        METHOD PUBLIC OVERRIDE MC_ReadAxisError
            VAR_INPUT
                AxisRef         :   AXOpen.Components.Abstractions.Drives.IAxoAxisReference;
                Enable          :   BOOL;                       //  Get the value of the parameter continuously while enabled
            END_VAR
            VAR_OUTPUT
                Valid           :   BOOL;                       //  A valid output is available at the method
                Busy            :   BOOL;                       //  The method is not finished and new output values are to be expected
                Error           :   BOOL;                       //  Signals that an error has occurred within the method
                ErrorID         :   DINT;                       //  Error identification
                AxisErrorID     :   DWORD;                      //  The value of the axis error. These values are vendor specific
            END_VAR
            VAR
                _AxisReference :  REF_TO AXOpen.Components.Rexroth.Drives.AxoCtrlxDriveXscAxisReference;
                _category  :   AXOpen.Messaging.eAxoMessageCategory;
            END_VAR

            _AxisReference ?= AxisRef;

            IF(_AxisReference = NULL) THEN
                Messenger.Activate(     UINT#1730, eAxoMessageCategory#ProgrammingError);
                DriveStatus.Error.Id := UINT#1730;
                RETURN;
            END_IF;

            IF Enable AND NOT MC_ReadAxisErrorEnable_PV AND _State = UINT#0 THEN
                _AxisReference^.Status.CurrentMotionTaskId := AXOpen.Components.Drives.eAxoMotionTaskId#Axo_ReadAxisError;
                _AxisReference^.Data.Cycle := _AxisReference^.Data.Cycle + ULINT#2;
                MC_ReadAxisErrorCycle := _AxisReference^.Data.Cycle ;
            END_IF;

            // IF Enable THEN
            //     THIS.UpdateInputs(_AxisReference^);
            //     IF _State = UINT#0 THEN
            //         Busy := TRUE;
            //         MC_ReadAxisErrorErrorID := WORD#16#0000;
            //         Parametrization.Inputs.Enable := FALSE;
            //         _State := UINT#310;
            //     END_IF;
            //     IF _State = UINT#310 THEN
            //         Busy := TRUE;
            //         Parametrization.Inputs.Enable := TRUE;
            //         Parametrization.Inputs.ReadWrite   := FALSE;
            //         Parametrization.Inputs.ParameterNo := 12306;
            //         Parametrization.Inputs.Subindex    := 0;
            //         Parametrization.Inputs.AxisNo  := BYTE#1;
            //         Parametrization.Inputs.HardwareId  := _AxisReference^.Data.hwIdModuleAccessPoint;
            //         IF Parametrization.Outputs.Done AND NOT Parametrization.Outputs.Error THEN
            //             MC_ReadAxisErrorValid := TRUE;
            //             MC_ReadAxisErrorValue := Parametrization.Outputs.ValueReadLINT;
            //             _State := UINT#311;
            //         END_IF;
            //         IF Parametrization.Outputs.Error THEN
            //             Messenger.Activate(         UINT#1731, eAxoMessageCategory#ProgrammingError);
            //             MC_ReadAxisErrorErrorID :=  WORD#1731;
            //             _State := UINT#319;
            //         END_IF;
            //     END_IF;
            //     IF _State = UINT#311 THEN
            //         Busy := TRUE;
            //         Parametrization.Inputs.Enable := FALSE;
            //         Parametrization.Inputs.ReadWrite   := FALSE;
            //         IF  NOT Parametrization.Outputs.Done THEN
            //             _State := UINT#310;
            //         END_IF;
            //     END_IF;
            //     IF _State = UINT#319 THEN
            //         Error := TRUE;
            //     END_IF;

            //     IF _State>=UINT#310 AND _State<UINT#317 THEN
            //         IF _AxisReference^.Data.Cycle <> MC_ReadAxisErrorCycle THEN
            //             _AxisReference^.Data.Cycle := _AxisReference^.Data.Cycle - ULINT#1;
            //             _State := UINT#319;
            //         END_IF;
            //     END_IF;
            //     THIS.UpdateOutputs(_AxisReference^);
            // END_IF;

            IF NOT Enable AND MC_ReadAxisErrorEnable_PV  THEN
                _AxisReference^.Status.CurrentMotionTaskId := AXOpen.Components.Drives.eAxoMotionTaskId#Axo_None;
                MC_ReadAxisErrorErrorID := WORD#0;
                MC_ReadAxisErrorCycle := ULINT#0;
                MC_ReadAxisErrorValid := FALSE;
                MC_ReadAxisErrorValue := LINT#0;
                _State := UINT#0;
            END_IF;

            ErrorID := TO_DINT(MC_ReadAxisErrorErrorID);
            Valid := MC_ReadAxisErrorValid;
            MC_ReadAxisErrorEnable_PV := Enable;

            Messenger.ActivateOnCondition(LastMessageCode,Enable AND Valid AND LastMessageCode = TO_ULINT(MC_ReadAxisErrorValue), eAxoMessageCategory#Error);
            // IF NOT Messenger.IsActive THEN
            IF Messenger.MessengerState = eAxoMessengerState#Idle THEN
                LastMessageCode := TO_ULINT(MC_ReadAxisErrorValue);
            END_IF;
        END_METHOD

        ///<summary>
        /// This method makes the transition from the State ‘ErrorStop’ to ‘Standstill’ or ‘Disabled’ by resetting all
        /// internal axis-related errors – it does not affect the output of the other methods.
        ///</summary>
        VAR INTERNAL
            MC_ResetState       : 	UINT := UINT#0;
            MC_ResetPower_PV    : 	BOOL := FALSE;
        END_VAR
        METHOD PUBLIC OVERRIDE MC_Reset
            VAR_INPUT
                AxisRef         :   AXOpen.Components.Abstractions.Drives.IAxoAxisReference;
                Execute         :   BOOL;                       //  Resets all internal axis-related error
            END_VAR
            VAR_OUTPUT
                Done            :   BOOL;                       //  ‘Standstill’ or ‘Disabled’_State is reached
                Busy            :   BOOL;                       //  The method is not finished and new output values are to be expected
                Error           :   BOOL;                       //  Signals that an error has occurred within the method
                ErrorID         :   DINT;                       //  Error identification
            END_VAR
            VAR
                _AxisReference :  REF_TO AXOpen.Components.Rexroth.Drives.AxoCtrlxDriveXscAxisReference;
            END_VAR

            _AxisReference ?= AxisRef;

            IF(_AxisReference = NULL) THEN
                Messenger.Activate(     UINT#1740, eAxoMessageCategory#ProgrammingError);
                DriveStatus.Error.Id := UINT#1740;
                RETURN;
            END_IF;

            IF Execute THEN
                IF Execute AND MC_ResetState = UINT#0 THEN
                    IF AxoPower_Task.IsSwitchedOn() OR
                       _AxisReference^.Outputs.DriveControlWord_S_0_0134_0_0.DriveEnable OR
                       _AxisReference^.Outputs.DriveControlWord_S_0_0134_0_0.DriveOn THEN
                         MC_ResetPower_PV := TRUE;
                    END_IF;
                    IF MC_ResetPower_PV THEN
                        MC_ResetState   := UINT#1;
                    ELSE
                        MC_ResetState   := UINT#10;
                    END_IF;
                END_IF;

                IF MC_ResetState = UINT#1 THEN
                    Busy := TRUE;
                    THIS.AxoPower_Task.Manual();
                    THIS.AxoPower_Task.SwitchOff();
                    IF THIS.AxoPower_Task.IsSwitchedOff() THEN
                        MC_ResetState := UINT#10;
                    END_IF;
                END_IF;

                IF MC_ResetState = UINT#10 THEN
                    IF MC_ResetPower_PV THEN
                        THIS.AxoPower_Task.Manual();
                        THIS.AxoPower_Task.SwitchOff();
                    END_IF;
                    Done            := FALSE;
                    Busy            := TRUE;
                    Error           := FALSE;
                    ErrorID         := UINT#0;
                    _AxisReference^.Outputs.SignalControlWord_S_0_0145_0_0.AcceptanceOfPositioningCommandValue := FALSE;
                    _AxisReference^.Outputs.SignalControlWord_S_0_0145_0_0.HomingControl := FALSE;
                    _AxisReference^.Outputs.SignalControlWord_S_0_0145_0_0.AbsoluteRelative := FALSE;
                    _AxisReference^.Outputs.SignalControlWord_S_0_0145_0_0.ImmediateChange := TRUE;
                    _AxisReference^.Outputs.SignalControlWord_S_0_0145_0_0.JogPositive := FALSE;
                    _AxisReference^.Outputs.SignalControlWord_S_0_0145_0_0.JogNegative := FALSE;
                    _AxisReference^.Outputs.SignalControlWord_S_0_0145_0_0.ClearError := TRUE;
                    IF NOT _AxisReference^.Inputs.DriveStatusWord_S_0_0135_0_0.DriveErrorZKL1 THEN
                        MC_ResetState := UINT#20;
                    END_IF;
                END_IF;

                IF MC_ResetState = UINT#20 THEN
                    Done            := FALSE;
                    Busy            := TRUE;
                    Error           := FALSE;
                    ErrorID         := UINT#0;
                    _AxisReference^.Outputs.SignalControlWord_S_0_0145_0_0.ClearError := FALSE;
                    IF NOT _AxisReference^.Inputs.DriveStatusWord_S_0_0135_0_0.DriveErrorZKL1 THEN
                        IF MC_ResetPower_PV THEN
                            MC_ResetState   := UINT#21;
                        ELSE
                            MC_ResetState   := UINT#30;
                        END_IF;
                    END_IF;
                END_IF;

                IF MC_ResetState = UINT#21 THEN
                    THIS.AxoPower_Task.Manual();
                    THIS.AxoPower_Task.SwitchOn();
                    Busy := TRUE;
                    IF THIS.AxoPower_Task.IsSwitchedOn() THEN
                        MC_ResetState := UINT#30;
                    END_IF;

                END_IF;

                IF MC_ResetState = UINT#30 THEN
                    MC_ResetPower_PV := FALSE;
                    Done            := TRUE;
                    Busy            := FALSE;
                    Error           := FALSE;
                    ErrorID         := UINT#0;
                END_IF;
            END_IF;
            IF NOT Execute THEN
                Done := FALSE;
                Error:=FALSE;
                ErrorID := DINT#0;
                Busy := FALSE;
                _AxisReference^.Outputs.SignalControlWord_S_0_0145_0_0.ClearError := FALSE;
                MC_ResetState := UINT#0;
            END_IF;
        END_METHOD

        METHOD PUBLIC OVERRIDE Restore
            MC_HomeExecute_PV					:= FALSE;
            MC_HomeErrorID					    := DINT#0;
            MC_HomeCycle					    := ULINT#0;
            MC_StopExecute_PV					:= FALSE;
            MC_StopErrorID					    := DINT#0;
            MC_StopCycle					    := ULINT#0;
            MC_HaltExecute_PV					:= FALSE;
            MC_HaltErrorID					    := DINT#0;
            MC_HaltCycle					    := ULINT#0;
            MC_MoveAbsoluteExecute_PV			:= FALSE;
            MC_MoveAbsoluteErrorID				:= DINT#0;
            MC_MoveAbsoluteCycle				:= ULINT#0;
            MC_MoveAbsoluteContinuousUpdate_SV  := FALSE;
            MC_MoveAbsolutePosition_PV          := LREAL#0.0;
            MC_MoveAbsoluteVelocity_PV          := LREAL#0.0;
            MC_MoveAbsoluteAcceleration_PV      := LREAL#0.0;
            MC_MoveAbsoluteDeceleration_PV      := LREAL#0.0;
            MC_MoveAbsoluteJerk_PV              := LREAL#0.0;
            MC_MoveAbsoluteDirection_PV         := AXOpen.Components.Abstractions.Drives.eAxoDriveDirection#CurrentDirection;
            MC_MoveRelativeExecute_PV			:= FALSE;
            MC_MoveRelativeErrorID				:= DINT#0;
            MC_MoveRelativeCycle				:= ULINT#0;
            MC_MoveRelativeContinuousUpdate_SV  := FALSE;
            MC_MoveRelativeDistance_PV          := LREAL#0.0;
            MC_MoveRelativeVelocity_PV          := LREAL#0.0;
            MC_MoveRelativeAcceleration_PV      := LREAL#0.0;
            MC_MoveRelativeDeceleration_PV      := LREAL#0.0;
            MC_MoveRelativeJerk_PV              := LREAL#0.0;
            MC_MoveAdditiveExecute_PV			:= FALSE;
            MC_MoveAdditiveErrorID				:= DINT#0;
            MC_MoveAdditiveCycle				:= ULINT#0;
            MC_MoveAdditiveContinuousUpdate_SV  := FALSE;
            MC_MoveAdditiveDistance_PV          := LREAL#0.0;
            MC_MoveAdditiveVelocity_PV          := LREAL#0.0;
            MC_MoveAdditiveAcceleration_PV      := LREAL#0.0;
            MC_MoveAdditiveDeceleration_PV      := LREAL#0.0;
            MC_MoveAdditiveJerk_PV              := LREAL#0.0;
            MC_MoveVelocityExecute_PV			:= FALSE;
            MC_MoveVelocityErrorID				:= WORD#0;
            MC_MoveVelocityCycle				:= ULINT#0;
            MC_MoveVelocityContinuousUpdate_SV  := FALSE;
            MC_MoveVelocityVelocity_PV          := LREAL#0.0;
            MC_MoveVelocityAcceleration_PV      := LREAL#0.0;
            MC_MoveVelocityDeceleration_PV      := LREAL#0.0;
            MC_MoveVelocityJerk_PV              := LREAL#0.0;
            MC_MoveVelocityDirection_PV         := AXOpen.Components.Abstractions.Drives.eAxoDriveDirection#CurrentDirection;
            MC_TorqueControlExecute_PV			:= FALSE;
            MC_TorqueControlErrorID				:= DINT#0;
            MC_TorqueControlCycle				:= ULINT#0;
            MC_TorqueControlContinuousUpdate_SV := FALSE;
            MC_TorqueControlTorque_PV           := LREAL#0.0;
            MC_TorqueControlTorqueRamp_PV       := LREAL#0.0;
            MC_TorqueControlPositionLimit_PV    := LREAL#0.0;
            MC_TorqueControlVelocity_PV         := LREAL#0.0;
            MC_TorqueControlAcceleration_PV     := LREAL#0.0;
            MC_TorqueControlDeceleration_PV     := LREAL#0.0;
            MC_TorqueControlJerk_PV             := LREAL#0.0;
            MC_TorqueControlDirection_PV        := AXOpen.Components.Abstractions.Drives.eAxoDriveDirection#CurrentDirection;
            MC_SetPositionExecute_PV			:= FALSE;
            MC_SetPositionErrorID				:= DINT#0;
            MC_SetPositionCycle					:= ULINT#0;
            MC_SetPositionActualPosition        := LINT#0;
            MC_ReadParameterEnable_PV           := FALSE;
            MC_ReadParameterErrorID             := DINT#0;
            MC_ReadParameterCycle			    := ULINT#0;
            MC_ReadParameterValue			    := LINT#0;
            MC_ReadParameterValid			    := FALSE;
            MC_ReadRealParameterEnable_PV       := FALSE;
            MC_ReadRealParameterErrorID         := DINT#0;
            MC_ReadRealParameterCycle			:= ULINT#0;
            MC_ReadRealParameterValue			:= REAL#0.0;
            MC_ReadRealParameterValid			:= FALSE;
            MC_ReadBoolParameterEnable_PV       := FALSE;
            MC_ReadBoolParameterErrorID         := WORD#0;
            MC_ReadBoolParameterCycle			:= ULINT#0;
            MC_ReadBoolParameterValue			:= FALSE;
            MC_ReadBoolParameterValid			:= FALSE;
            MC_WriteParameterExecute_PV         := FALSE;
            MC_WriteParameterErrorID            := WORD#0;
            MC_WriteParameterCycle			    := ULINT#0;
            MC_WriteRealParameterExecute_PV     := FALSE;
            MC_WriteRealParameterErrorID        := WORD#0;
            MC_WriteRealParameterCycle			:= ULINT#0;
            MC_WriteBoolParameterExecute_PV     := FALSE;
            MC_WriteBoolParameterErrorID        := WORD#0;
            MC_WriteBoolParameterCycle			:= ULINT#0;
            MC_ReadDigitalInputEnable_PV        := FALSE;
            MC_ReadDigitalInputErrorID          := WORD#0;
            MC_ReadDigitalInputCycle			:= ULINT#0;
            MC_ReadDigitalInputValue			:= FALSE;
            MC_ReadDigitalInputValid			:= FALSE;
            MC_ReadDigitalOutputEnable_PV       := FALSE;
            MC_ReadDigitalOutputErrorID         := WORD#0;
            MC_ReadDigitalOutputCycle			:= ULINT#0;
            MC_ReadDigitalOutputValue			:= FALSE;
            MC_ReadDigitalOutputValid			:= FALSE;
            MC_WriteDigitalOutputExecute_PV     := FALSE;
            MC_WriteDigitalOutputErrorID        := WORD#0;
            MC_WriteDigitalOutputCycle			:= ULINT#0;
            MC_ReadStatusEnable_PV				:= FALSE;
            MC_ReadStatusDone_PV				:= FALSE;
            MC_ReadStatusStateNumber			:= INT#0;
            MC_ReadMotionStateEnable_PV         := FALSE;
            MC_ReadMotionStateErrorID           := WORD#0;
            MC_ReadMotionStateCycle			    := ULINT#0;
            MC_ReadMotionStateValue			    := LINT#0;
            MC_ReadMotionStateValid			    := FALSE;
            MC_ReadAxisErrorEnable_PV           := FALSE;
            MC_ReadAxisErrorErrorID             := WORD#0;
            MC_ReadAxisErrorCycle			    := ULINT#0;
            MC_ReadAxisErrorValue			    := LINT#0;
            MC_ReadAxisErrorValid			    := FALSE;
            LastMessageCode                     := ULINT#0;
            MC_ResetState                       := UINT#0;
            AxisRefExt.Data.Cycle               := ULINT#0;
            _State                              := UINT#0;
            DriveStatus.Action.Id := UINT#0;
            DriveStatus.Error.Id  := UINT#0;
            Messenger.Restore();
            TaskMessenger.Restore();

            //AxoPower_Task.Restore();
            AxoStop_Task.Restore();
            AxoHalt_Task.Restore();
            AxoHome_Task.Restore();
            AxoMoveAbsolute_Task.Restore();
            AxoMoveRelative_Task.Restore();
            AxoMoveAdditive_Task.Restore();
            AxoMoveVelocity_Task.Restore();
            AxoTorqueControl_Task.Restore();
            AxoSetPosition_Task.Restore();
            AxoSetOverride_Task.SwitchOff();
            AxoReadParameter_Task.SwitchOff();
            AxoReadRealParameter_Task.SwitchOff();
            AxoReadBoolParameter_Task.SwitchOff();
            AxoWriteParameter_Task.Restore();
            AxoWriteRealParameter_Task.Restore();
            AxoWriteBoolParameter_Task.Restore();
            AxoReadDigitalInput_Task.SwitchOff();
            AxoReadDigitalOutput_Task.SwitchOff();
            AxoWriteDigitalOutput_Task.Restore();
            AxoReadActualPosition_Task.SwitchOff();
            AxoReadActualVelocity_Task.SwitchOff();
            AxoReadActualTorque_Task.SwitchOff();
            AxoReadStatus_Task.SwitchOff();
            AxoReadMotionState_Task.SwitchOff();
            AxoReadAxisInfo_Task.SwitchOff();
            AxoReadAxisError_Task.SwitchOff();
            AxoReset_Task.Restore();
            AxoJogPositive.RemoteSwitchOn := FALSE;
            AxoJogPositive.StartMotion := FALSE;
            AxoJogPositive.StopMotion := FALSE;
            AxoJogNegative.RemoteSwitchOn := FALSE;
            AxoJogNegative.StartMotion := FALSE;
            AxoJogNegative.StopMotion := FALSE;

            // AxisRefExt.Outputs.CommandPosition_S_0_0282_0_0 := DINT#0;
            // AxisRefExt.Outputs.CommandVelocity_S_0_0259_0_0 := DINT#0;
            // AxisRefExt.Outputs.CommandAcceleration_S_0_0260_0_0 := DINT#0;
            // AxisRefExt.Outputs.CommandDecceleration_S_0_0359_0_0 := DINT#0;
            // AxisRefExt.Outputs.CommandTorque_S_0_0080_0_0 := INT#0;

            SUPER.Restore();

            RestoreTask.DoneWhen(TRUE);
        END_METHOD
        METHOD PRIVATE CallTimers
            VAR_INPUT
                signal : BOOL;
            END_VAR

            _infoTimer.OnDelay(THIS, signal AND DriveConfig.InfoTime > LT#0S ,DriveConfig.InfoTime);
            _errorTimer.OnDelay(THIS, signal AND DriveConfig.ErrorTime > LT#0S , DriveConfig.ErrorTime);
        END_METHOD
        METHOD PRIVATE CallTimers
            VAR_INPUT
                signal_1 : BOOL;
                signal_2 : BOOL;
            END_VAR

            _infoTimer.OnDelay(THIS, signal_1 AND DriveConfig.InfoTime > LT#0S ,DriveConfig.InfoTime);
            _errorTimer.OnDelay(THIS, signal_2 AND DriveConfig.ErrorTime > LT#0S , DriveConfig.ErrorTime);
        END_METHOD
    END_CLASS
END_NAMESPACE
